// TIA Portal V19 export
TYPE "LAF_typeDevDiagStructGetDiag"
TITLE = Structure GETDIAG / Struktur GETDIAG
// This data type contains the structure of instruction GETDIAG / PN device Diagnose
// stored: Access Published
   STRUCT
      mode { ExternalAccessible := 'False'; ExternalVisible := 'False'; ExternalWritable := 'False'} : UInt := 0;   // Mode: 0-DWord, 1-DIS, 2-DNN / Mode: 1-DIS, 2-DNN
      laddr { ExternalAccessible := 'False'; ExternalVisible := 'False'; ExternalWritable := 'False'} : HW_IO;   // Use "DevHWAddr_HWTYPE5_PNIF / HWTYPE = 5 (Submodul_PROFINET_Interface)" / use "DevHWAddr_HWTYPE5_PNIF / HWTYPE = 5 (Submodul_PROFINET_Interface)"
      retVal { ExternalAccessible := 'False'; ExternalVisible := 'False'; ExternalWritable := 'False'} : Int;   // Return value
      cntDiag { ExternalAccessible := 'False'; ExternalVisible := 'False'; ExternalWritable := 'False'} : UInt := 0;   // Reserviert (immer 0) / Reserved (always 0)
      diagDataMode0 { ExternalAccessible := 'False'; ExternalVisible := 'False'; ExternalWritable := 'False'} : DWord;   // Diagnostic information / Diagnose Information
      diagDataMode1 { ExternalAccessible := 'False'; ExternalVisible := 'False'; ExternalWritable := 'False'} : DIS;   // Diagnostic information (not in use) / Diagnose Information (z.Zt. nicht in Verwendung)
      diagDataMode2 { ExternalAccessible := 'False'; ExternalVisible := 'False'; ExternalWritable := 'False'} : DNN;   // Diagnostic information / Diagnose Information
      detailData { ExternalAccessible := 'False'; ExternalVisible := 'False'; ExternalWritable := 'False'} : UInt;   // Not in use / Nicht in Verwendung
   END_STRUCT;
END_TYPE
